// TwinCAT 3 PLC project Untitled1
// ProgramVersion: 3.1.4026.21
// libraries:
//   Tc2_Standard, * (Beckhoff Automation GmbH)
//   Tc2_System, * (Beckhoff Automation GmbH)
// project tree:
//   / PlcTask.TcTTO, TestPrg.TcPOU
//   POUs/WorkThrough/ DoublePneumaticActuator.TcPOU, ITF_LiftActuator.TcIO, PneumaticActuator.TcPOU, LiftManager.TcPOU
//   POUs/ MAIN.TcPOU
// real-time tasks:
//   TASK PlcTask: cycle T#10ms, priority 20, ADS port 350

CONFIGURATION Untitled1
    RESOURCE PLC ON TwinCAT3
        TASK PlcTask(INTERVAL := T#10ms, PRIORITY := 20);
        PROGRAM MAIN WITH PlcTask : MAIN;
    END_RESOURCE
END_CONFIGURATION

// ---- POUs/WorkThrough/ITF_LiftActuator.TcIO
INTERFACE ITF_LiftActuator

METHOD ExtendActuator : BOOL
VAR_INPUT
END_VAR
END_METHOD

METHOD RetractActuator : BOOL
VAR_INPUT
END_VAR
END_METHOD

END_INTERFACE

// ---- POUs/MAIN.TcPOU
PROGRAM MAIN
VAR
	// This is Sebastien's Edit 1 from 64
	// yet another comment
	
	myPneumaticPusher : PneumaticActuator(UnitMaxOperatingPressure := 100000.0, UnitMinOperatingPressure := 5000.0);
	iState: INT;
	EnableSystemLogging: BOOL;
	DisableLoggingSystem: BOOL;
	mySecondPneumaticPusher: DoublePneumaticActuator (UnitMaxOperatingPressure := 100000.0, UnitMinOperatingPressure := 5000.0);
	control: INT;
	liftManager : LiftManager := (MyLiftActuator := myPneumaticPusher);
	
END_VAR


CASE control OF 
	1: 
		liftManager.MyLiftActuator := myPneumaticPusher;
		control := 0;
	2:	
		liftManager.MyLiftActuator := mySecondPneumaticPusher;
		control := 0;
END_CASE

liftManager.Cycle();

IF EnableSystemLogging THEN
	EnableSystemLogging := FALSE;
	myPneumaticPusher.SetLogginState := TRUE;
END_IF

IF DisableLoggingSystem THEN
	DisableLoggingSystem := FALSE;
	myPneumaticPusher.SetLogginState := FALSE;
END_IF

TestPrg();

END_PROGRAM

// ---- POUs/WorkThrough/PneumaticActuator.TcPOU
FUNCTION_BLOCK PneumaticActuator IMPLEMENTS ITF_LiftActuator

VAR
	extendOutput AT %Q* : BOOL;
	retractOutput AT %Q* : BOOL;
	_MaxOperatingPressure: LREAL;
	_MinOperatingPressure: LREAL;
	_logging: BOOL;
END_VAR

METHOD ExtendActuator : BOOL
VAR_INPUT
END_VAR
ExtendActuator := TRUE; // return value
extendOutput := TRUE; // IO
retractOutput := FALSE; // IO
IF _logging THEN
	SendTraceData('Extending.....');
END_IF
END_METHOD

//FB_Init is always available implicitly and it is used primarily for initialization.
//The return value is not evaluated. For a specific influence, you can also declare the
//methods explicitly and provide additional code there with the standard initialization
//code. You can evaluate the return value.
METHOD FB_Init: BOOL
VAR_INPUT
    bInitRetains: BOOL; // TRUE: the retain variables are initialized (reset warm / reset cold)
    bInCopyCode: BOOL;  // TRUE: the instance will be copied to the copy code afterward (online change)   
	UnitMaxOperatingPressure	: LREAL;
	UnitMinOperatingPressure	: LREAL;
END_VAR
_MaxOperatingPressure := UnitMaxOperatingPressure;
_MinOperatingPressure := UnitMinOperatingPressure;
END_METHOD

PROPERTY MaxOperatingPressure : LREAL
GET
MaxOperatingPressure := _MaxOperatingPressure;
END_GET
END_PROPERTY

PROPERTY MinOperatingPressure : LREAL
GET
MinOperatingPressure := _MinOperatingPressure;
END_GET
END_PROPERTY

METHOD RetractActuator : BOOL
VAR_INPUT
END_VAR
RetractActuator := TRUE;
extendOutput := FALSE;
retractOutput := TRUE;
IF _logging THEN
	SendTraceData('Retracting.....');
END_IF
END_METHOD

METHOD PROTECTED SendTraceData : BOOL
VAR_INPUT
	MessageToSend	: STRING(80);
END_VAR
ADSLOGSTR(msgCtrlMask	:= ADSLOG_MSGTYPE_LOG,
			msgFmtStr	:= MessageToSend,
			strArg		:= '');
END_METHOD

PROPERTY PUBLIC SetLogginState : BOOL
GET
SetLogginState := _logging;
END_GET
SET
_logging := SetLogginState;
END_SET
END_PROPERTY

END_FUNCTION_BLOCK

// ---- POUs/WorkThrough/DoublePneumaticActuator.TcPOU
FUNCTION_BLOCK DoublePneumaticActuator EXTENDS PneumaticActuator

VAR
	extendOutput1 AT %Q* : BOOL;
	retractOutput1 AT %Q* : BOOL;
END_VAR

METHOD ExtendActuator : BOOL
extendOutput1 := TRUE;
retractOutput1 := FALSE;

SUPER^.ExtendActuator();
END_METHOD

METHOD RetractActuator : BOOL
RetractActuator := TRUE;
extendOutput := FALSE;
extendOutput1 := FALSE;
retractOutput := TRUE;
retractOutput1 := TRUE;

IF _logging THEN
	SendTraceData('Retracting...');
END_IF
END_METHOD

END_FUNCTION_BLOCK

// ---- POUs/WorkThrough/LiftManager.TcPOU
{attribute 'no_explicit_call' := 'Do not call this POU directly'}
FUNCTION_BLOCK LiftManager

VAR
	_myLiftActuator : ITF_LiftActuator;
	
	iState: INT;
END_VAR

METHOD Cycle : BOOL
VAR_INPUT
END_VAR
CASE iState OF 	

	1:
		_myLiftActuator.ExtendActuator();
		iState := 0;
	2:
		_myLiftActuator.RetractActuator();
		iState := 0;
END_CASE
END_METHOD

PROPERTY MyLiftActuator : ITF_LiftActuator
GET
END_GET
SET
END_SET
END_PROPERTY

END_FUNCTION_BLOCK

// ---- TestPrg.TcPOU
PROGRAM TestPrg
VAR
END_VAR

TC_EVENTS.ST_Warning.event1;
TC_EVENTS.ST_Warning.ST_WarningEvent3;
TC_EVENTS.ST_Warning.ST_WarningEvent4;
TC_EVENTS.ST_Warning.ST_WarningEvent5;
//TC_EVENTS.ST_Warning.ST_WarningEvent6;
TC_EVENTS.ST_Warning.ST_WarningEvent61;
TC_EVENTS.ST_Warning.OneWeirdEvent;

END_PROGRAM
